{attribute 'linkalways'} 
{attribute 'no_explicit_call' := 'This FB is a CLASS and must be accessed using methods or properties'}
{attribute 'enable_dynamic_creation'}
FUNCTION_BLOCK FeedTableCommand EXTENDS Command
VAR
	_nci : I_Nci;
	_fb : REFERENCE TO FB_NciFeedTable;
	_table : I_Table;
	_null : ST_NciFeedGroupTable;
END_VAR

METHOD CleanUp
_fb(
	bExecute := FALSE,
	bReset := FALSE,
	stNciToPlc := _nci._InternalNciPlcRef.nciToPlc,
	stFeedGroupTable := _null
);
END_METHOD

METHOD FB_init : BOOL
VAR_INPUT
	bInitRetains : BOOL; // if TRUE, the retain variables are initialized (warm start / cold start)
	bInCopyCode : BOOL;  // if TRUE, the instance afterwards gets moved into the copy code (online change)
	nci : I_Nci;
	fb : REFERENCE TO FB_NciFeedTable;
	table : I_Table;
END_VAR
IF nci <> 0 THEN
	nci := nci;
END_IF

IF __ISVALIDREF(fb) THEN
	_fb REF= fb;
END_IF

IF table <> 0 THEN
	_table := table;
END_IF
END_METHOD

METHOD PROTECTED OnAbort
VAR_INPUT
	CommandState : I_CommandAbortingState;
END_VAR
CleanUp();
END_METHOD

METHOD PROTECTED  WhileBusy
VAR_INPUT
	CommandState : I_CommandBusyState;
END_VAR
_fb(
	bExecute := TRUE,
	bReset := FALSE,
	stNciToPlc := _nci._InternalNciPlcRef.nciToPlc,
	stFeedGroupTable := _table._InternalTable,
);

IF NOT _fb.bFeedBusy THEN
	RETURN;
END_IF

IF _fb.bError THEN
	CleanUp();
	CommandState.SetError(_fb.nErrorId);
	RETURN;
END_IF

CleanUp();

CommandState.SetDOne();
END_METHOD

END_FUNCTION_BLOCK

(* stored: Version 1.1.0.1, ProductVersion 3.1.4024.12
   POU FeedTableCommand: Id {47449ea4-f3a6-4cd2-ad0d-de8d8af22b7e}, SpecialFunc None
   Method CleanUp: Id {047e7829-343c-4868-91e4-b3d7d4faa214}
   Method FB_init: Id {64023528-108f-4dd7-b70d-71b580ccf5bb}
   Method OnAbort: Id {67b2f407-3231-4886-b77a-843fc7e83188}
   Method WhileBusy: Id {5a186f95-98b6-4199-8ba9-6ff883d335f1} *)
